TYPE U16 : UINT; END_TYPE

(* stored: Version 1.1.0.1
   DUT U16: Id {c9da0d8f-eb00-022f-1220-a05acfb48868} *)
